FUNCTION_BLOCK E_D_FF (* Basic Function Block Type *)
  (* Standard: 61499-2 *)
  (* Version 0.0, 9/9/2026, macie, Schneider Electric, Template *)
  PACKAGE Main;
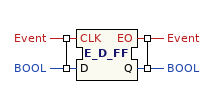
  EVENT_INPUT
    CLK WITH D; (* Initialization Request *)
  END_EVENT
  EVENT_OUTPUT
    EO WITH Q; (* Initialization Confirm *)
  END_EVENT
  VAR_INPUT
    D : BOOL := FALSE; (* Input event qualifier *)
  END_VAR
  VAR_OUTPUT
    Q : BOOL := FALSE; (* Output event qualifier *)
  END_VAR
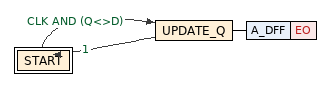
  EC_STATES
    START; (* Initial State *)
    UPDATE_Q : A_DFF -> EO;
  END_STATES
  EC_TRANSITIONS
    START TO UPDATE_Q := CLK AND (Q<>D);
    UPDATE_Q TO START := 1;
  END_TRANSITIONS
  ALGORITHM A_DFF IN ST: (* Normally executed algorithm *)
;
Q:=D;
  END_ALGORITHM
END_FUNCTION_BLOCK
